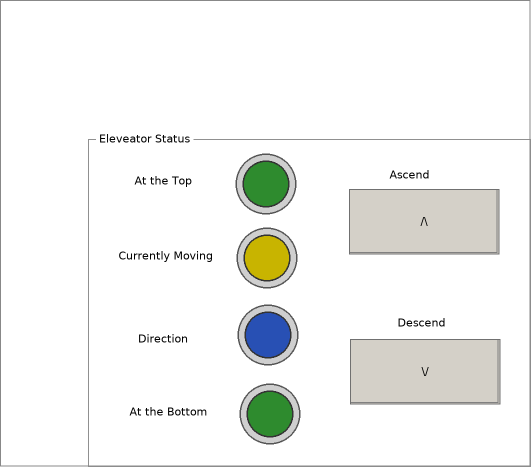
VISUALIZATION Q7_V  // 531x467
    GroupBox (88,131 443x336), "Eleveator Status"
        Lamp1 (143,18 70x70), style: Lamp-Lamp1-Green
        Lamp1 (144,92 70x70), variable: Q7.moving, style: Lamp-Lamp1-Yellow
        Lamp1 (145,169 70x70), variable: true, style: Lamp-Lamp1-Blue
        Lamp1 (147,248 70x70), style: Lamp-Lamp1-Green
        Button (261,58 150x65), "/\"
            OnMouseClick: execute { Q7.button_up := TRUE }
        Button (262,208 150x65), "\/"
        Label (286,177 95x30), "Descend"
        Label (277,29 89x30), "Ascend"
        Label (25,193 100x30), "Direction"
        Label (29,266 103x30), "At the Bottom"
        Label (27,35 97x30), "At the Top"
        Label (25,110 106x30), "Currently Moving"
END_VISUALIZATION

(* stored: Version 1.1.0.1, ProductVersion 3.1.4024.12
   Visu Q7_V: Id {e6be822e-650a-47e9-bc7b-59f4d5ae5266} *)
